// TIA Portal V20 export
FUNCTION_BLOCK "ComRF160B"   // FB182, SCL
TITLE = ComRF160B
{ S7_Optimized_Access := 'TRUE' }
AUTHOR : DIL
VERSION : 1.0
// stored: MemoryReserve 100, SetENOAutomatically false
   VAR_INPUT
      enable { ExternalAccessible := 'False'; ExternalVisible := 'False'; ExternalWritable := 'False'} : Bool;
      cont { ExternalAccessible := 'False'; ExternalVisible := 'False'; ExternalWritable := 'False'} : Bool;
      localPort { ExternalAccessible := 'False'; ExternalVisible := 'False'; ExternalWritable := 'False'} : UInt := 2000;   // local UDP/TCP port number
      interfaceId { ExternalAccessible := 'False'; ExternalVisible := 'False'; ExternalWritable := 'False'} : HW_ANY := 16#0040;
      connectionId { ExternalAccessible := 'False'; ExternalVisible := 'False'; ExternalWritable := 'False'} : CONN_OUC := 16#0001;
   END_VAR
   VAR_OUTPUT
      error { ExternalAccessible := 'False'; ExternalVisible := 'False'; ExternalWritable := 'False'} : Bool;
      done { ExternalAccessible := 'False'; ExternalVisible := 'False'; ExternalWritable := 'False'} : Bool;
      connected { ExternalAccessible := 'False'; ExternalVisible := 'False'; ExternalWritable := 'False'} : Bool;
      restart { ExternalAccessible := 'False'; ExternalVisible := 'False'; ExternalWritable := 'False'} : Bool;
      lenEpcId { ExternalAccessible := 'False'; ExternalVisible := 'False'; ExternalWritable := 'False'} : Byte;
      lenData { ExternalAccessible := 'False'; ExternalVisible := 'False'; ExternalWritable := 'False'} : Byte;
      status { ExternalAccessible := 'False'; ExternalVisible := 'False'; ExternalWritable := 'False'} : Word;
      statusId { ExternalAccessible := 'False'; ExternalVisible := 'False'; ExternalWritable := 'False'} : UInt;
   END_VAR
   VAR_IN_OUT
      reset { ExternalAccessible := 'False'; ExternalVisible := 'False'; ExternalWritable := 'False'} : Bool;
      data : Variant;
      epcId : Variant;
   END_VAR
   VAR
      statConnectionData { ExternalAccessible := 'False'; ExternalVisible := 'False'; ExternalWritable := 'False'; S7_SetPoint := 'True'} : TCON_IP_v4;
      instTRCV { ExternalAccessible := 'False'; ExternalVisible := 'False'; ExternalWritable := 'False'; S7_SetPoint := 'True'} : TRCV_C;
      statRCV { ExternalAccessible := 'False'; ExternalVisible := 'False'; ExternalWritable := 'False'} : Struct
         Enable : Bool;
         Cont : Bool;
         Len : UDInt;
         Done : Bool;
         Busy : Bool;
         Error : Bool;
         Status : Word;
         RcvLen : UDInt;
         DataValues : Array[0..311] of Byte;
         COM_RST : Bool;
         ADDR : Bool;
      END_STRUCT;
      statErrorRcv { ExternalAccessible := 'False'; ExternalVisible := 'False'; ExternalWritable := 'False'} : Bool;
      statLastErrorStatus { ExternalAccessible := 'False'; ExternalVisible := 'False'; ExternalWritable := 'False'} : Word;
      statBufferPtr { ExternalAccessible := 'False'; ExternalVisible := 'False'; ExternalWritable := 'False'} : UDInt;
      statRCVBufferValues { ExternalAccessible := 'False'; ExternalVisible := 'False'; ExternalWritable := 'False'} : Array[0..1000] of Byte;
   END_VAR
   VAR_TEMP
      tempBufferInitValues : Array[0..1000] of Byte;
      tempBufferTelValues : Array[0..311] of Byte;
      tempBufferValues : Array[0..1000] of Byte;
      tempStatus : Word;
      tempDataReceived : Bool;
      tempTelegramComplete : Bool;
      tempRetValue : Int;
      tempLenEpcID : Byte;
      tempLenData : Byte;
      tempSize : UDInt;
      tempRcvLen : UDInt;
      tempEpcIdLen : UDInt;
      tempUserDataLen : UDInt;
      tempError : Bool;
      tempLoop : Int;
      tempDataValid : Bool;
      tempRestart : Bool;
      tempTelegramValid : Bool;
      tempStatusId : UInt;
   END_VAR
   VAR CONSTANT
      TELEGRAM_LEN : UInt := 312;
      BUFFER_LEN : UInt := 1000;
      POS_DATA_LEN : UInt := 130;
      POS_EPC_ID_LEN : UInt := 1;
      ZERO : UInt;
      MAX_DATA_LEN : UInt := 182;
      MAX_EPC_ID_LEN : UInt := 128;
   END_VAR
BEGIN
   //=============================================================================
   // Siemens AG
   // (c)Copyright 2022 All Rights Reserved
   //-----------------------------------------------------------------------------
   // Library: ---
   // Tested with: S7-1511-1 PN, FW V2.9
   // Engineering: TIA Portal V18 
   // Restrictions: --
   // Requirements: To be used only with a Profinet Interface and RF160 mobile
   //               reader.
   // Functionality: Connect to a RF160 mobile reader and receive EPC-ID/UID and data
   //                send by the mobile reader. TCP (Ad-hoc mode) mode will be
   //                used for establishing a communication connection.
   //-----------------------------------------------------------------------------
   //
   // Change log table:
   // Version  Date       Expert in charge Changes applied
   // 01.00.00 01.09.2022 Meierhofer Simon First released version
   //=============================================================================

   //===========================================================
   // Init
   //===========================================================
   #statConnectionData.InterfaceId := #interfaceId;
   #statConnectionData.ID := #connectionId;
   #statConnectionData.LocalPort := #localPort;
   #statRCV.Enable := #enable;
   #statRCV.Cont := #cont;

   //===========================================================
   // connection
   //===========================================================
   #instTRCV(EN_R := #statRCV.Enable,
             CONT := #statRCV.Cont,
             LEN := #statRCV.Len,
             ADHOC := True,
             DONE => #statRCV.Done,
             BUSY => #statRCV.Busy,
             ERROR => #statRCV.Error,
             STATUS => #statRCV.Status,
             RCVD_LEN => #statRCV.RcvLen,
             DATA := #statRCV.DataValues,
             ADDR := #statRCV.ADDR,
             COM_RST := #statRCV.COM_RST,
             CONNECT := #statConnectionData);

   #tempStatusId := 4;
   #tempStatus := #statRCV.Status;
   #statErrorRcv := #statRCV.Error;
   #tempDataReceived := NOT #statRCV.Busy AND NOT #statRCV.Error AND #statRCV.Done;
   #connected := (#statRCV.Status = 16#7004) OR (#statRCV.Status = 16#7006);


   IF #statErrorRcv THEN
     #tempError := true;
     #tempStatus := #statRCV.Status;
   ELSE
     #statRCV.COM_RST := False;
   END_IF;

   //===========================================================
   // copy received data to main buffer
   //===========================================================
   IF #tempDataReceived AND NOT #statErrorRcv AND NOT #reset THEN

     #tempDataValid := (#statRCV.RcvLen <> 16#0001) AND (#statRCV.DataValues[0] <> 16#01);

     //check bufferoverflow
     IF #tempDataValid THEN
       IF #statRCV.RcvLen + #statBufferPtr < #BUFFER_LEN THEN
         #tempRcvLen := #statRCV.RcvLen;
         #tempTelegramComplete := false;

         // move data to static buffer
         MOVE_BLK(IN := #statRCV.DataValues[0],
                  COUNT := #tempRcvLen,
                  OUT => #statRCVBufferValues[#statBufferPtr]);
         #statBufferPtr := #statBufferPtr + #tempRcvLen;
       ELSE
         #tempStatus := 16#8D13;
         #tempStatusId := 1;
       END_IF;

     END_IF;
   END_IF;

   //===========================================================
   // split data to telegram(312 bytes) and main buffer
   //===========================================================
   IF #statBufferPtr >= #TELEGRAM_LEN AND
     NOT #statErrorRcv AND NOT #reset THEN

     //1. copy to temp buffer
     MOVE_BLK(IN := #statRCVBufferValues[0],
              COUNT := #BUFFER_LEN,
              OUT => #tempBufferValues[0]);

     //2.init main buffer
     MOVE_BLK(IN := #tempBufferInitValues[0],
              COUNT := #BUFFER_LEN,
              OUT => #statRCVBufferValues[0]);

     //3.create one telegram (first part)
     MOVE_BLK(IN := #tempBufferValues[0],
              COUNT := #TELEGRAM_LEN,
              OUT => #tempBufferTelValues[0]);

     //4. move the remaning data back to main buffer (second part)
     MOVE_BLK(IN := #tempBufferValues[TELEGRAM_LEN],
              COUNT := #BUFFER_LEN - #TELEGRAM_LEN,
              OUT => #statRCVBufferValues[0]);

     //5. set poiter to the correct array(main) index
     #statBufferPtr := (#statBufferPtr - #TELEGRAM_LEN);

     // set flags
     #tempTelegramComplete := True;

     // verify Telegram
     IF #tempBufferTelValues[311] = 16#7E THEN
       #tempTelegramValid := true;
     ELSE
       #tempStatus := 16#8D12;
       #tempError := true;
       #tempStatusId := 1;
       GOTO Exception;
     END_IF;
   END_IF;

   //===========================================================
   // edit telegram 
   //===========================================================
   IF #tempTelegramComplete AND #tempTelegramValid
     AND NOT #statErrorRcv AND NOT #reset THEN

     #tempLenData := #tempBufferTelValues[POS_DATA_LEN];
     #tempLenEpcID := #tempBufferTelValues[POS_EPC_ID_LEN];
     #tempRestart := #tempBufferTelValues[ZERO] = 16#FF;

     //verification data array
     IF #tempLenData > #MAX_DATA_LEN THEN
       #tempStatus := 16#8D21;
       #tempStatusId := 1;
       #tempError := true;
       GOTO Exception;
     END_IF;

     //verification id array
     IF (#tempLenEpcID = #ZERO) AND (#tempRestart = false) THEN
       #tempStatus := 16#8D31;
       #tempStatusId := 1;
       #tempError := true;
       GOTO Exception;
     ELSIF #tempLenEpcID > #MAX_EPC_ID_LEN THEN
       #tempStatus := 16#8D32;
       #tempStatusId := 1;
       #tempError := true;
       GOTO Exception;
     END_IF;

     //===========================================================
     //EPC output
     //===========================================================
     #tempSize := CountOfElements(#epcId);


     IF #tempSize > #tempLenEpcID THEN
       IF #tempLenEpcID > #ZERO THEN
         #tempRetValue := MOVE_BLK_VARIANT(SRC := #tempBufferTelValues,
                                           SRC_INDEX := 2,
                                           COUNT := #tempLenEpcID,
                                           DEST => #epcId,
                                           DEST_INDEX := 0);

         IF #tempRetValue <> 0 THEN
           #tempStatus := INT_TO_WORD(#tempRetValue);
           #tempStatusId := 2;
           #tempError := true;
           GOTO Exception;
         END_IF;
       END_IF;
     ELSE
       #tempStatus := 16#8D14;
       #tempStatusId := 1;
       #tempError := True;
       GOTO Exception;
     END_IF;


     //===========================================================
     //Data output
     //===========================================================
     #tempSize := CountOfElements(#data);
     IF #tempSize > #tempLenData THEN
       IF #tempLenData > 0 THEN
         #tempRetValue := MOVE_BLK_VARIANT(SRC := #tempBufferTelValues,
                                           SRC_INDEX := 131,
                                           COUNT := #tempLenData,
                                           DEST => #data,
                                           DEST_INDEX := 0);

         IF #tempRetValue <> 0 THEN
           #tempStatus := INT_TO_WORD(#tempRetValue);
           #tempStatusId := 3;
           #tempError := true;
           GOTO Exception;
         END_IF;
       END_IF;

     ELSE
       #tempStatus := 16#8D24;
       #tempStatusId := 1;
       #tempError := true;
       GOTO Exception;
     END_IF;

     #restart := #tempRestart;
     #lenData := #tempLenData;
     #lenEpcId := #tempLenEpcID;
     #done := true;

     //status
     IF (#tempLenEpcID = #ZERO) AND (#tempRestart = true) THEN
       #tempStatus := 16#7002;
     ELSE
       #tempStatus := 16#7001;
     END_IF;

     #tempStatusId := 1;
   ELSE

     #restart := false;
     #lenData := 0;
     #lenEpcId := 0;
     #done := false;

     //===========================================================
     // Reset EPC-ID output
     //=========================================================== 
     #tempRetValue := MOVE_BLK_VARIANT(SRC := #tempBufferInitValues,
                                       SRC_INDEX := 0,
                                       COUNT := CountOfElements(#epcId),
                                       DEST => #epcId,
                                       DEST_INDEX := 0);

     IF #tempRetValue <> #ZERO THEN
       #tempStatus := INT_TO_WORD(#tempRetValue);
       #tempStatusId := 5;
       #tempError := true;
       GOTO Exception;
     END_IF;

     //===========================================================
     // Reset #DATA output
     //=========================================================== 
     #tempRetValue := MOVE_BLK_VARIANT(SRC := #tempBufferInitValues,
                                       SRC_INDEX := 0,
                                       COUNT := CountOfElements(#data),
                                       DEST => #data,
                                       DEST_INDEX := 0);

     IF #tempRetValue <> #ZERO THEN
       #tempStatus := INT_TO_WORD(#tempRetValue);
       #tempStatusId := 6;
       #tempError := true;
       GOTO Exception;
     END_IF;

   END_IF;

   //===========================================================
   //reset
   //===========================================================
   IF #reset THEN

     //init rcv data
     MOVE_BLK(IN := #tempBufferInitValues[0],
              COUNT := #TELEGRAM_LEN,
              OUT => #statRCV.DataValues[0]);

     //init rcv buffer
     MOVE_BLK(IN := #tempBufferInitValues[0],
              COUNT := #BUFFER_LEN,
              OUT => #statRCVBufferValues[0]);

     #statBufferPtr := 0;
     #statLastErrorStatus := 0;
     #tempRcvLen := 0;

     //===========================================================
     // Reset EPC-ID output
     //=========================================================== 
     #tempRetValue := MOVE_BLK_VARIANT(SRC := #tempBufferInitValues,
                                       SRC_INDEX := 0,
                                       COUNT := CountOfElements(#epcId),
                                       DEST => #epcId,
                                       DEST_INDEX := 0);
     IF #tempRetValue <> 0 THEN
       #tempStatus := INT_TO_WORD(#tempRetValue);
       #tempStatusId := 7;
     END_IF;

     #lenEpcId := 0;

     //===========================================================
     // Reset #DATA output
     //=========================================================== 
     #tempRetValue := MOVE_BLK_VARIANT(SRC := #tempBufferInitValues,
                                       SRC_INDEX := 0,
                                       COUNT := CountOfElements(#data),
                                       DEST => #data,
                                       DEST_INDEX := 0);
     IF #tempRetValue <> 0 THEN
       #tempStatus := INT_TO_WORD(#tempRetValue);
       #tempStatusId := 8;
     END_IF;

     #lenData := 0;

     //Output

     #reset := False;
   END_IF;

   Exception:
   IF #tempError THEN
     IF #tempStatus = 16#80C4 THEN

       #tempStatus:= 16#7002;
       #error := false;

     ELSE
       #statLastErrorStatus := #tempStatus;
       #error := true;
     END_IF;
   ELSE
     #error := False;
   END_IF;

   #status := #tempStatus;
   #statusId := #tempStatusId;
END_FUNCTION_BLOCK
